Staubli VAL3: empty1dNum.pgx

public program empty1dNum(num& x_nNum[])
  local num l_nIndex
begin

  //empty a 1d array of num

  for l_nIndex=0 to size(x_nNum)-1
      x_nNum[l_nIndex]=0
  endFor

end
